FUNCTION_BLOCK ProductOrder
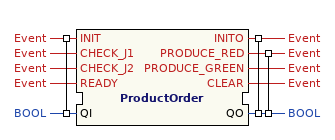
  EVENT_INPUT
    INIT WITH QI;
    CHECK_J1;
    CHECK_J2;
    READY;
  END_EVENT
  EVENT_OUTPUT
    INITO WITH QO;
    PRODUCE_RED WITH QO;
    PRODUCE_GREEN;
    CLEAR;
  END_EVENT
  VAR_INPUT
    QI : BOOL;
  END_VAR
  VAR_OUTPUT
    QO : BOOL;
  END_VAR
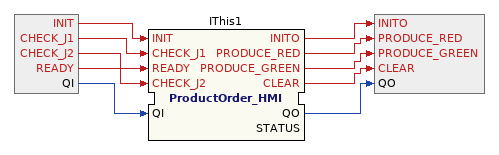
  FBS
    IThis1 : ProductOrder_HMI;
  END_FBS
  EVENT_CONNECTIONS
    INIT TO IThis1.INIT;
    CHECK_J1 TO IThis1.CHECK_J1;
    READY TO IThis1.READY;
    IThis1.INITO TO INITO;
    IThis1.PRODUCE_RED TO PRODUCE_RED;
    IThis1.PRODUCE_GREEN TO PRODUCE_GREEN;
    IThis1.CLEAR TO CLEAR;
    CHECK_J2 TO IThis1.CHECK_J2;
  END_CONNECTIONS
  DATA_CONNECTIONS
    QI TO IThis1.QI;
    IThis1.QO TO QO;
  END_CONNECTIONS
END_FUNCTION_BLOCK
